TYPE T_CodeRSKU : STRING[9];
END_TYPE

(* stored: Version 1.1.0.1
   DUT T_CodeRSKU: Id {7927ffe6-e972-49cd-aa84-bc1095157dcb} *)
